(*This block implements interface "IOopExmpl" 
	>>this means is must have the methods described in the interface

*)
FUNCTION_BLOCK OopExmplRandomObjectWithInterface IMPLEMENTS IOopExmpl
VAR
	HM_b1:BOOL; //not used for example
END_VAR

//code we are not using in the interface example
HM_b1:=TRUE;
//...
//...
//...
//...
//...

//Method the object must implement because of the interface
METHOD MustHaveMethod : BOOL
VAR_INPUT
	I:BOOL;
END_VAR
MustHaveMethod := I;
END_METHOD

END_FUNCTION_BLOCK

(* stored: Version 1.1.0.1
   POU OopExmplRandomObjectWithInterface: Id {69daf245-9213-0e4a-2208-af7cea4de983}, SpecialFunc None
   Method MustHaveMethod: Id {55cbf681-63ec-0fb4-37b1-c79d8d7c158e} *)
